FUNCTION_BLOCK TurnTable
VAR_INPUT
	EN   : BOOL;
	iStartCW    	:  BOOL;    // Clockwise Move Command 
	iStartCCW   	:  BOOL;    // Counterclockwise Move Command 
	iFwdPosSensor  	:  BOOL;    // Forward Position sensor 180* feedback
	iRevPosSensor  	:  BOOL;    // Forward Position sensor 0* feedback
END_VAR
VAR_OUTPUT
	Eno  : BOOL;
	qMotorRun  :  BOOL ; 	// Motor Run Status
	qMotorDir  :  BOOL ;    // Motor Direction Status 
END_VAR
VAR
END_VAR

// Motor Safety
IF  iStartCW AND iStartCCW THEN
	qMotorRun := FALSE;
	qMotorDir := FALSE;
END_IF

// TURNTABLE OPERATION
	IF iStartCW AND NOT iFwdPosSensor THEN
		qMotorRun := TRUE;
		qMotorDir := FALSE;
	ELSIF iStartCCW AND NOT iRevPosSensor THEN
		qMotorRun := TRUE;
		qMotorDir := TRUE;
		ELSE 
		qMotorRun := FALSE;
		qMotorDir := FALSE;
	END_IF

END_FUNCTION_BLOCK

(* stored: Version 1.1.0.1, ProductVersion 3.1.4024.16
   POU TurnTable: Id {0c8caac1-1793-446a-9a6b-e8732c18542f}, SpecialFunc None *)
